% RSLogix 500 project horizontal_tank_integer_running.RSS, saved by version 8.30.00.16 %
PROJECT "UNTITLED"    % processor: Bul.1763 MicroLogix 1100 Series A %

PROGRAM FILES
  LAD 2   2 rungs
  LAD 255 "ONEDEPTH"  10 rungs

DATA FILES
  O0 OUTPUT  4 elements
  I1 INPUT  6 elements
  S2 STATUS  66 elements
  B3 BINARY  1 elements
  T4 TIMER  1 elements
  C5 COUNTER  1 elements
  R6 CONTROL  1 elements
  N7 INTEGER  20 elements
  F8 FLOAT  1 elements
  F254   128 elements
  N255   256 elements

LADDER 2
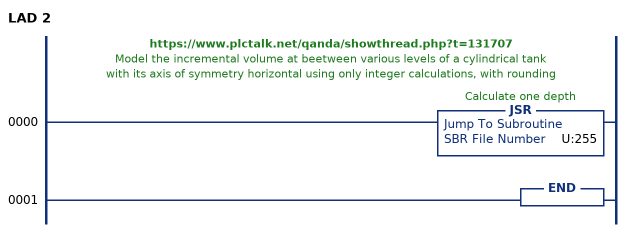
% Rung: 0 %
% TITLE: https://www.plctalk.net/qanda/showthread.php?t=131707 %
% Model the incremental volume at beetween various levels of a cylindrical tank
% with its axis of symmetry horizontal using only integer calculations, with rounding %
SOR JSR U:255 EOR
%   U:255  "Calculate one depth" %
% Rung: 1 %
SOR END EOR

LADDER 255 "ONEDEPTH"
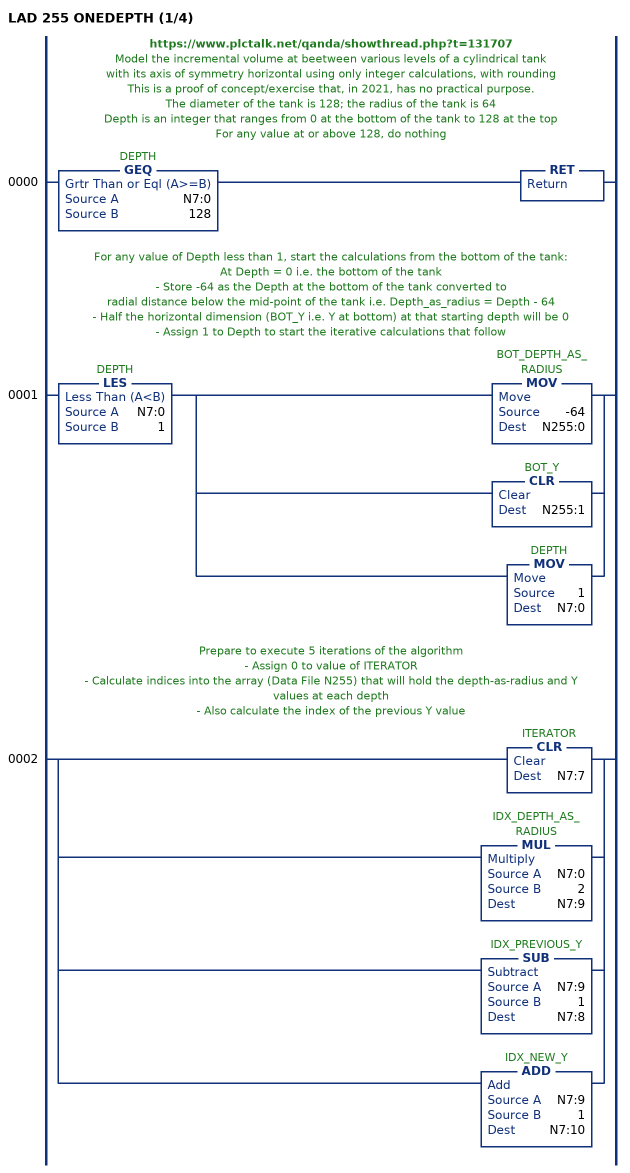
% Rung: 0 %
% TITLE: https://www.plctalk.net/qanda/showthread.php?t=131707 %
% Model the incremental volume at beetween various levels of a cylindrical tank
% with its axis of symmetry horizontal using only integer calculations, with rounding
% 
% This is a proof of concept/exercise that, in 2021, has no practical purpose.
% 
% The diameter of the tank is 128; the radius of the tank is 64
% Depth is an integer that ranges from 0 at the bottom of the tank to 128 at the top
% For any value at or above 128, do nothing %
SOR GEQ N7:0 128 RET EOR
%   N7:0  DEPTH %
% Rung: 1 %
% For any value of Depth less than 1, start the calculations from the bottom of the tank:
% At Depth = 0 i.e. the bottom of the tank
% - Store -64 as the Depth at the bottom of the tank converted to
%   radial distance below the mid-point of the tank i.e. Depth_as_radius = Depth - 64
% - Half the horizontal dimension (BOT_Y i.e. Y at bottom) at that starting depth will be 0
% - Assign 1 to Depth to start the iterative calculations that follow %
SOR LES N7:0 1 BST MOV -64 N255:0 NXB CLR N255:1 NXB MOV 1 N7:0 BND EOR
%   N7:0  DEPTH %
%   N255:0  BOT_DEPTH_AS_RADIUS %
%   N255:1  BOT_Y %
% Rung: 2 %
% Prepare to execute 5 iterations of the algorithm
% - Assign 0 to value of ITERATOR
% - Calculate indices into the array (Data File N255) that will hold the depth-as-radius and Y values at each depth
% - Also calculate the index of the previous Y value %
SOR BST CLR N7:7 NXB MUL N7:0 2 N7:9 NXB SUB N7:9 1 N7:8 NXB ADD N7:9 1 N7:10 BND EOR
%   N7:7  ITERATOR %
%   N7:0  DEPTH %
%   N7:9  IDX_DEPTH_AS_RADIUS %
%   N7:8  IDX_PREVIOUS_Y %
%   N7:10  IDX_NEW_Y %

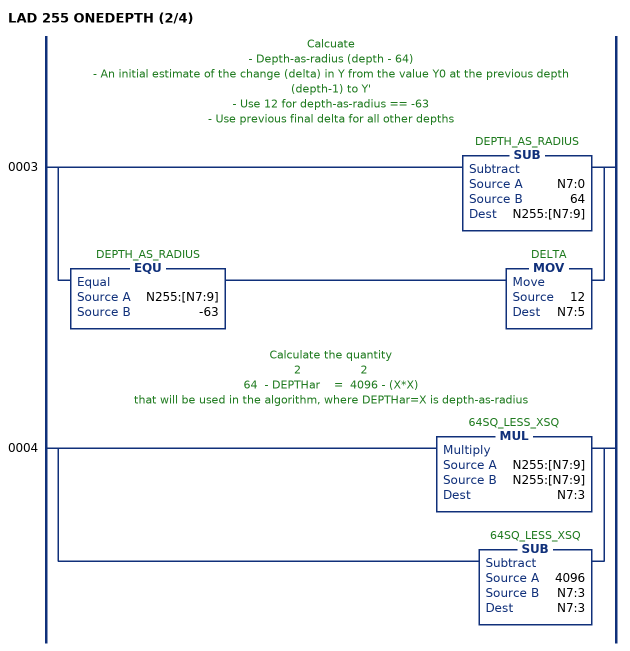
% Rung: 3 %
% Calcuate
% - Depth-as-radius (depth - 64)
% - An initial estimate of the change (delta) in Y from the value Y0 at the previous depth (depth-1) to Y'
%   - Use 12 for depth-as-radius == -63
%   - Use previous final delta for all other depths %
SOR BST SUB N7:0 64 N255:[N7:9] NXB EQU N255:[N7:9] -63 MOV 12 N7:5 BND EOR
%   N7:0  DEPTH %
%   N255:[N7:9]  DEPTH_AS_RADIUS %
%   N7:9  IDX_DEPTH_AS_RADIUS %
%   N7:5  DELTA %
% Rung: 4 %
% Calculate the quantity
% 
%      2                 2
%   64  - DEPTHar    =  4096 - (X*X)
% 
% that will be used in the algorithm, where DEPTHar=X is depth-as-radius %
SOR BST MUL N255:[N7:9] N255:[N7:9] N7:3 NXB SUB 4096 N7:3 N7:3 BND EOR
%   N255:[N7:9]  DEPTH_AS_RADIUS %
%   N7:9  IDX_DEPTH_AS_RADIUS %
%   N7:3  64SQ_LESS_XSQ %

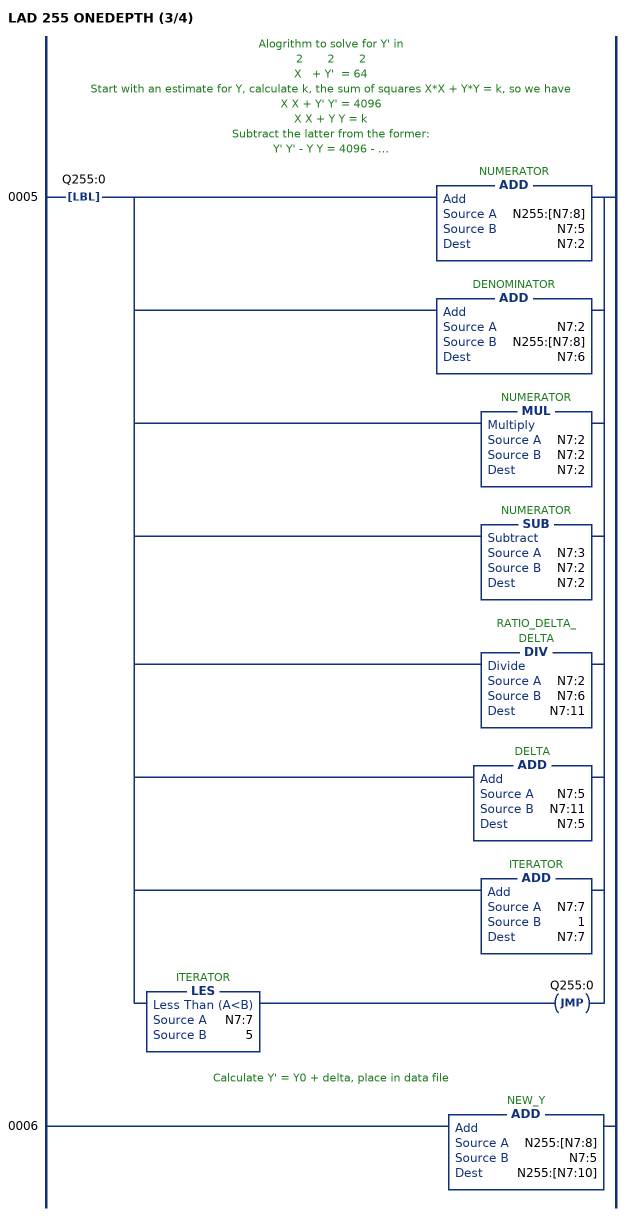
% Rung: 5 %
% Alogrithm to solve for Y' in
%       2       2       2
%     X   + Y'  = 64
% Start with an estimate for Y, calculate k, the sum of squares X*X + Y*Y = k, so we have
%    X X + Y' Y' = 4096
%    X X + Y Y = k
% Subtract the latter from the former:
%    Y' Y' - Y Y = 4096 - k
% Assume there is a difference, delta, between Y' and Y:
%   Y' = Y + delta
% Substituting
%   (Y+delta) (Y+delta) - Y Y = 4096 - k
%   Y Y + 2 Y delta + delta delta - Y*Y = 4096 - k
%   2  Y delta + delta delta = 4096 - k
%   delta (2Y + delta) = 4096 - k
%   delta = (4096 - k) / (2Y + deltaOLD)
% Use successive substitution:
% - Start with an estimate of Y as the Y0 from the previous depth,
% - Use the previous depth's delta as deltaOLD, so Y' = Y0 + deltaOLD, to calculate an incremental delta:
%   incrdelta = (4096 - k) / (2Y + deltaOLD)
% - Increment deltaOLD by incrdelta to get a new deltaOLD
%   deltaOLD = deltaOLD + incrdelta = deltaOLD + (4096 - k) / (2Y + deltaOLD)
% and repeat for five iterations %
SOR LBL Q255:0 BST ADD N255:[N7:8] N7:5 N7:2 NXB ADD N7:2 N255:[N7:8] N7:6 NXB MUL N7:2 N7:2 N7:2 NXB SUB N7:3 N7:2 N7:2 NXB DIV N7:2 N7:6 N7:11 NXB ADD N7:5 N7:11 N7:5 NXB ADD N7:7 1 N7:7 NXB LES N7:7 5 JMP Q255:0 BND EOR
%   N255:[N7:8]  PREVIOUS_Y %
%   N7:8  IDX_PREVIOUS_Y %
%   N7:5  DELTA %
%   N7:2  NUMERATOR %
%   N7:6  DENOMINATOR %
%   N7:3  64SQ_LESS_XSQ %
%   N7:11  RATIO_DELTA_DELTA %
%   N7:7  ITERATOR %
% Rung: 6 %
% Calculate Y' = Y0 + delta, place in data file %
SOR ADD N255:[N7:8] N7:5 N255:[N7:10] EOR
%   N255:[N7:8]  PREVIOUS_Y %
%   N7:8  IDX_PREVIOUS_Y %
%   N7:5  DELTA %
%   N255:[N7:10]  NEW_Y %
%   N7:10  IDX_NEW_Y %

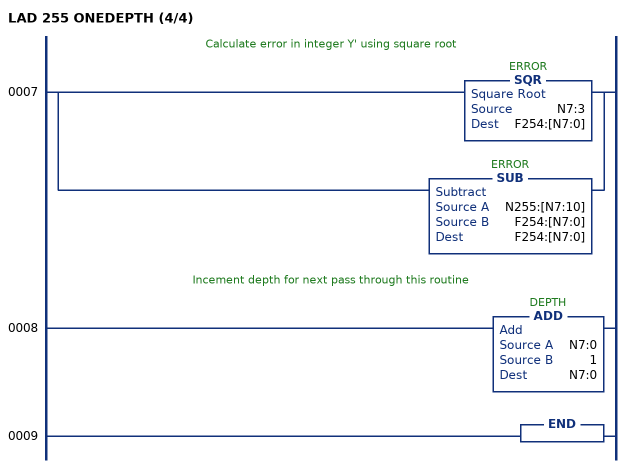
% Rung: 7 %
% Calculate error in integer Y' using square root %
SOR BST SQR N7:3 F254:[N7:0] NXB SUB N255:[N7:10] F254:[N7:0] F254:[N7:0] BND EOR
%   N7:3  64SQ_LESS_XSQ %
%   F254:[N7:0]  ERROR %
%   N7:0  DEPTH %
%   N255:[N7:10]  NEW_Y %
%   N7:10  IDX_NEW_Y %
% Rung: 8 %
% Incement depth for next pass through this routine %
SOR ADD N7:0 1 N7:0 EOR
%   N7:0  DEPTH %
% Rung: 9 %
SOR END EOR

OTHER DOCUMENTED ADDRESSES
  N7:4  RADIUS

DATA TABLE (non-zero values as saved)
DATA B3
% B3:0 % 0X0001
DATA N7
% N7:0 % 128 0 6 127 0 -5 27 5 253 254
% N7:10 % 255 0 0 0 0 0 0 0 0 0
DATA F254
% F254:0 % 0 -0.2694273 0.1254921 -0.3649158 -0.2710571
% F254:5 % 0.2008057 -0.05549812 -0.1032639 0.01613235 0.2738647
% F254:10 % -0.3511276 0.1252174 -0.3095169 0.3347702 0.05002975
% F254:15 % -0.1703758 -0.3320198 -0.4396133 0.5028076 0.4917603
% F254:20 % -0.4757996 -0.4025307 -0.2907867 -0.1426506 0.04001617
% F254:25 % 0.2555428 -0.4975739 -0.2206841 0.08497238 0.4182854
% F254:30 % -0.2217674 0.1638794 -0.4256248 0.008930206 0.4668236
% F254:35 % -0.05260849 0.4500198 -0.02585602 -0.4807663 0.08480835
% F254:40 % -0.329586 0.2756348 -0.09991837 -0.4565964 0.205265
% F254:45 % -0.1146469 -0.4166107 0.2991104 0.03226471 -0.2173615
% F254:50 % -0.4499817 0.3342209 0.135067 -0.04759979 -0.2139244
% F254:55 % -0.3640289 0.5019684 0.3839645 0.2818718 0.19561
% F254:60 % 0.1251221 0.07035065 0.03125763 0.0078125 0
% F254:65 % 0.0078125 0.03125763 0.07035065 0.1251221 0.19561
% F254:70 % 0.2818718 0.3839645 -0.4980316 -0.3640289 -0.2139244
% F254:75 % -0.04759979 0.135067 0.3342209 -0.4499817 -0.2173615
% F254:80 % 0.03226471 0.2991104 -0.4166107 -0.1146469 0.205265
% F254:85 % -0.4565964 -0.09991837 0.2756348 -0.329586 0.08480835
% F254:90 % -0.4807663 -0.02585602 0.4500198 -0.05260849 0.4668236
% F254:95 % 0.008930206 -0.4256248 0.1638794 -0.2217674 0.4182854
% F254:100 % 0.08497238 -0.2206841 -0.4975739 0.2555428 0.04001617
% F254:105 % -0.1426506 -0.2907867 -0.4025307 -0.4757996 0.4917603
% F254:110 % 0.5028076 -0.4396133 -0.3320198 -0.1703758 0.05002975
% F254:115 % 0.3347702 -0.3095169 0.1252174 -0.3511276 0.2738647
% F254:120 % 0.01613235 -0.1032639 -0.05549812 0.2008057 -0.2710571
% F254:125 % -0.3649158 0.1254921 -0.2694273
DATA N255
% N255:0 % -64 0 -63 11 -62 16 -61 19 -60 22
% N255:10 % -59 25 -58 27 -57 29 -56 31 -55 33
% N255:20 % -54 34 -53 36 -52 37 -51 39 -50 40
% N255:30 % -49 41 -48 42 -47 43 -46 45 -45 46
% N255:40 % -44 46 -43 47 -42 48 -41 49 -40 50
% N255:50 % -39 51 -38 51 -37 52 -36 53 -35 54
% N255:60 % -34 54 -33 55 -32 55 -31 56 -30 57
% N255:70 % -29 57 -28 58 -27 58 -26 58 -25 59
% N255:80 % -24 59 -23 60 -22 60 -21 60 -20 61
% N255:90 % -19 61 -18 61 -17 62 -16 62 -15 62
% N255:100 % -14 62 -13 63 -12 63 -11 63 -10 63
% N255:110 % -9 63 -8 64 -7 64 -6 64 -5 64
% N255:120 % -4 64 -3 64 -2 64 -1 64 0 64
% N255:130 % 1 64 2 64 3 64 4 64 5 64
% N255:140 % 6 64 7 64 8 63 9 63 10 63
% N255:150 % 11 63 12 63 13 63 14 62 15 62
% N255:160 % 16 62 17 62 18 61 19 61 20 61
% N255:170 % 21 60 22 60 23 60 24 59 25 59
% N255:180 % 26 58 27 58 28 58 29 57 30 57
% N255:190 % 31 56 32 55 33 55 34 54 35 54
% N255:200 % 36 53 37 52 38 51 39 51 40 50
% N255:210 % 41 49 42 48 43 47 44 46 45 46
% N255:220 % 46 45 47 43 48 42 49 41 50 40
% N255:230 % 51 39 52 37 53 36 54 34 55 33
% N255:240 % 56 31 57 29 58 27 59 25 60 22
% N255:250 % 61 19 62 16 63 11
